(* PLC project Modbus, Beremiz Beremiz 1 *)
(* stored: creationDateTime 2018-07-27T13:19:12, modificationDateTime 2024-03-05T04:07:35 *)

PROGRAM program0
  VAR
    isensor AT %IX100.0.0.0 : BOOL;
    oconvey AT %QX100.0.1.0 : BOOL;
    isenor1 AT %IX100.0.2.1 : BOOL;
    oconvey1 AT %QX100.0.3.1 : BOOL;
  END_VAR

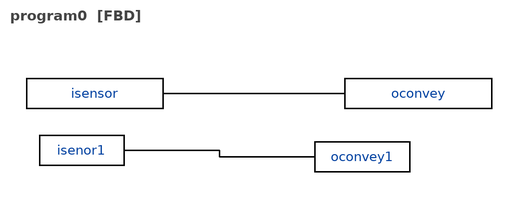
(* FBD diagram, written out as Structured Text *)
oconvey := isensor;
oconvey1 := isenor1;
END_PROGRAM

CONFIGURATION config
  RESOURCE resource1 ON PLC
    TASK task0(INTERVAL := T#20ms, PRIORITY := 0);
    PROGRAM instance0 WITH task0 : program0;
  END_RESOURCE
END_CONFIGURATION
